TYPE ST_ProcessData :
STRUCT
	batch		: STRING(100);
	number		: STRING(100);
	name		: STRING(100);
	value1		: REAL; 
	value2		: REAL;
	value3		: REAL;
	value4		: REAL;
	value5 		: REAL;
	value6		: REAL; 
END_STRUCT
END_TYPE

(* stored: Version 1.1.0.1, ProductVersion 3.1.4026.13
   DUT ST_ProcessData: Id {3d4f24af-b6dc-46ab-9964-91ccef45caf1} *)
